PROGRAM MAIN
VAR
END_VAR

END_PROGRAM

(* stored: Version 1.1.0.1, ProductVersion 3.1.4024.12
   POU MAIN: Id {5bcef741-3b68-077d-3d3e-300308b277da}, SpecialFunc None *)
